% RSLogix 500 project Bottle_Filling Process.RSS, saved by version 8.30.00.16 %
PROJECT "UNTITLED"    % processor: Bul.1763 MicroLogix 1100 Series B %

PROGRAM FILES
  LAD 2   7 rungs

DATA FILES
  O0 OUTPUT  4 elements
  I1 INPUT  6 elements
  S2 STATUS  66 elements
  B3 BINARY  1 elements
  T4 TIMER  1 elements
  C5 COUNTER  1 elements
  R6 CONTROL  1 elements
  N7 INTEGER  1 elements
  F8 FLOAT  1 elements

LADDER 2
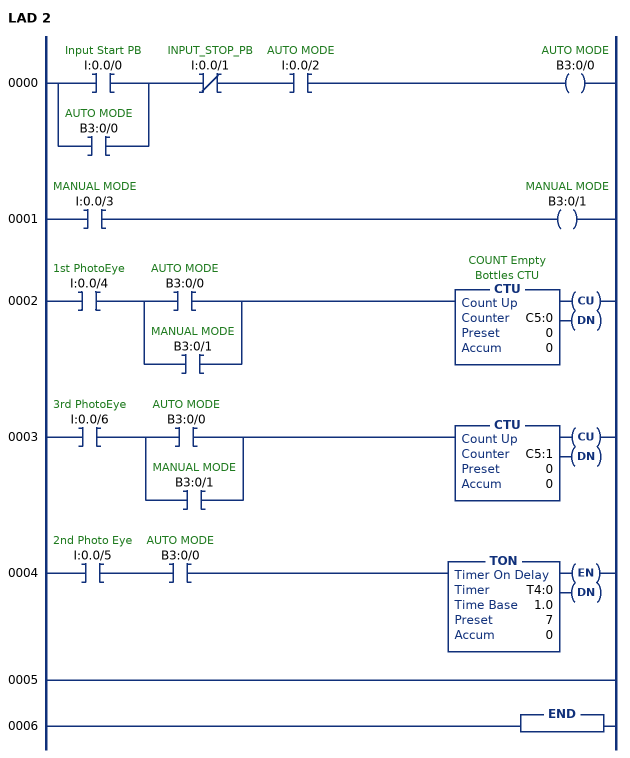
% Rung: 0 %  % edit flag set %
SOR BST XIC I:0.0/0 NXB XIC B3:0/0 BND XIO I:0.0/1 XIC I:0.0/2 OTE B3:0/0 EOR
%   I:0.0/0  "Input Start PB" %
%   B3:0/0  "AUTO MODE" %
%   I:0.0/1  INPUT_STOP_PB %
%   I:0.0/2  "AUTO MODE" %
% Rung: 1 %  % edit flag set %
SOR XIC I:0.0/3 OTE B3:0/1 EOR
%   I:0.0/3  "MANUAL MODE" %
%   B3:0/1  "MANUAL MODE" %
% Rung: 2 %  % edit flag set %
SOR XIC I:0.0/4 BST XIC B3:0/0 NXB XIC B3:0/1 BND CTU C5:0 0 0 EOR
%   I:0.0/4  "1st PhotoEye" %
%   B3:0/0  "AUTO MODE" %
%   B3:0/1  "MANUAL MODE" %
%   C5:0  CTU  "COUNT Empty Bottles" %
% Rung: 3 %  % edit flag set %
SOR XIC I:0.0/6 BST XIC B3:0/0 NXB XIC B3:0/1 BND CTU C5:1 0 0 EOR
%   I:0.0/6  "3rd PhotoEye" %
%   B3:0/0  "AUTO MODE" %
%   B3:0/1  "MANUAL MODE" %
% Rung: 4 %  % edit flag set %
SOR XIC I:0.0/5 XIC B3:0/0 TON T4:0 1.0 7 0 EOR
%   I:0.0/5  "2nd Photo Eye" %
%   B3:0/0  "AUTO MODE" %
% Rung: 5 %  % edit flag set %
SOR EOR
% Rung: 6 %
SOR END EOR
